{attribute 'qualified_only'}
{attribute 'strict'}
TYPE E_SeqTransport :
(
	UNKNOWN := 0,

	TB_TO_INFEED,
	TB_AT_INFEED,

	TB_TO_CENTRING,
	TB_AT_CENTRING,

	TB_TO_DOCKING,
	TB_AT_DOCKING
);
END_TYPE

(* stored: Version 1.1.0.1, ProductVersion 3.1.4024.12
   DUT E_SeqTransport: Id {eaed0fb9-54d6-42ad-96a1-4f80392c5ed1} *)
